(*
SPDX-FileCopyrightText: © 2026 Oleksandr Tiutyk <trofimich@gmail.com>
SPDX-License-Identifier: MIT
License: https://opensource.org/license/mit
*)

(*!
<summary>Exposes whether an object is bound to its required IO data.</summary>
<description>
Binding operations and the required IO channels belong to the concrete device API.
</description>
*)

INTERFACE IIOBindable EXTENDS IObject

(*!
<summary>Reports whether the required IO bindings are present.</summary>
<description>
The concrete device defines which bindings are required. This status does not establish hardware health,
communication state or freshness of IO values.
</description>
*)

{attribute 'monitoring' := 'call'}
PROPERTY FINAL BoundToIO : BOOL
GET
END_GET
END_PROPERTY

END_INTERFACE

(* stored: Version 1.1.0.1
   Itf IIOBindable: Id {c613c159-795e-4dc7-ae41-ac2b019d9330}
   Property BoundToIO: Id {133b2262-01f7-4288-a1ea-ef2b55cbb091}
   Get Get: Id {2f0f600d-241e-4f54-a080-d5f424f7851e} *)
